TYPE 
	T_IoLink64ByteData : ARRAY[0..7] OF BYTE; 
END_TYPE

(* stored: Version 1.1.0.1, ProductVersion 3.1.4024.15
   DUT T_IoLink64ByteData: Id {1edf497a-597c-05f7-1315-a3e3d2b318be} *)
